// TIA Portal V18 export
TYPE "RCS_KeyenceSR1000_HMI"
   STRUCT
      Manual : Struct   // Manual
         Preset : Bool;   // Preset
         Trigger : Bool;   // Trigger
      END_STRUCT;
      Status : Struct   // Status
         Ready : Bool;   // Ready
         Busy : Bool;   // Busy
         Failure : Bool;   // Failure
         Complete : Bool;   // Complete
         ReadOk : Bool;   // ReadOk
         ReadNok : Bool;   // ReadNok
         TimeOut : Bool;   // TimeOut
         Error : Bool;   // Error
         ErrorCode : UInt;   // ErrorCode
         Sequence : Int;   // Sequence
         iReTriggerTimes : USInt;   // iReTriggerTimes
         CurrentLength : UInt;   // CurrentLength
         CurrentCode : String[128];   // CurrentCode
         LastCode : String[128];   // LastCode
      END_STRUCT;
      Indata : Struct   // Indata
         ReadComplete : Bool;   // ReadComplete
         ReadFailure : Bool;   // ReadFailure
         GeneralErrorCode : UInt;   // GeneralErrorCode
         ReadResultCode : UInt;   // ReadResultCode
         ResultDataSize : UInt;   // ResultDataSize
      END_STRUCT;
      Outdata : Struct   // Outdata
         ReadCompleteClear : Bool;   // ReadCompleteClear
         ErrorClear : Bool;   // ErrorClear
         ReadRequest : Bool;   // ReadRequest
      END_STRUCT;
   END_STRUCT;
END_TYPE
